FUNCTION_BLOCK FUNCTIONALITY_CONTROLLER (* Composite Function Block Type *)
  (* Standard: 61499-2 *)
  (* Version 1.0, 2019-04-04, adeel *)
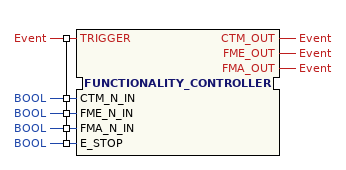
  EVENT_INPUT
    TRIGGER WITH CTM_N_IN, FME_N_IN, FMA_N_IN, E_STOP; (* Normal Execution Request *)
  END_EVENT
  EVENT_OUTPUT
    CTM_OUT; (* Execution Confirmation *)
    FME_OUT;
    FMA_OUT;
  END_EVENT
  VAR_INPUT
    CTM_N_IN : BOOL; (* Input event qualifier *)
    FME_N_IN : BOOL;
    FMA_N_IN : BOOL;
    E_STOP : BOOL;
  END_VAR
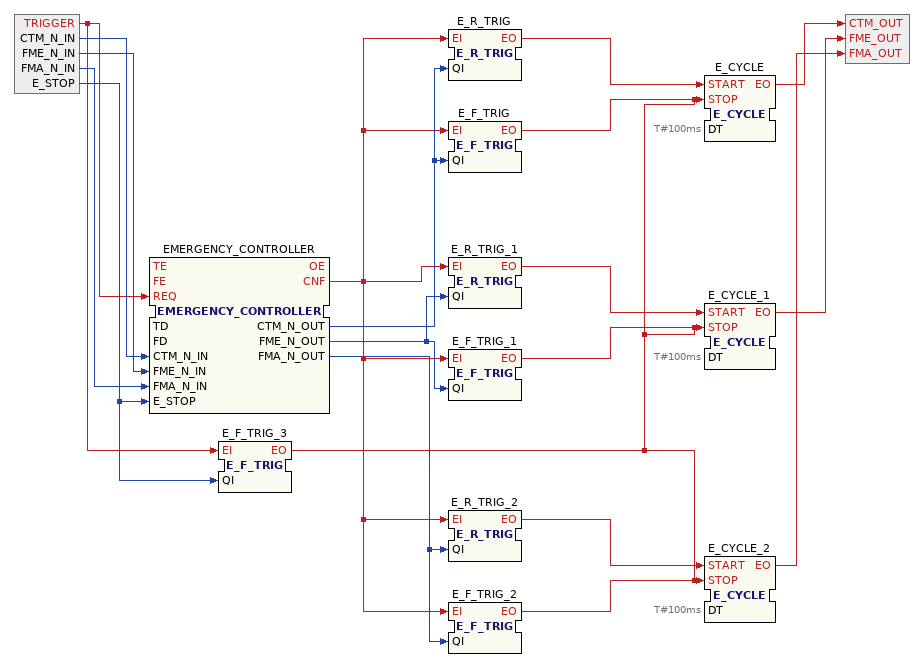
  FBS
    E_R_TRIG : E_R_TRIG;
    E_R_TRIG_1 : E_R_TRIG;
    E_R_TRIG_2 : E_R_TRIG;
    E_CYCLE : E_CYCLE(DT := T#100ms);
    E_CYCLE_1 : E_CYCLE(DT := T#100ms);
    E_CYCLE_2 : E_CYCLE(DT := T#100ms);
    E_F_TRIG : E_F_TRIG;
    E_F_TRIG_1 : E_F_TRIG;
    E_F_TRIG_2 : E_F_TRIG;
    EMERGENCY_CONTROLLER : EMERGENCY_CONTROLLER;
    E_F_TRIG_3 : E_F_TRIG;
  END_FBS
  EVENT_CONNECTIONS
    E_R_TRIG.EO TO E_CYCLE.START;
    E_F_TRIG.EO TO E_CYCLE.STOP;
    E_CYCLE.EO TO CTM_OUT;
    E_R_TRIG_1.EO TO E_CYCLE_1.START;
    E_F_TRIG_1.EO TO E_CYCLE_1.STOP;
    E_CYCLE_1.EO TO FME_OUT;
    E_R_TRIG_2.EO TO E_CYCLE_2.START;
    E_F_TRIG_2.EO TO E_CYCLE_2.STOP;
    E_CYCLE_2.EO TO FMA_OUT;
    EMERGENCY_CONTROLLER.CNF TO E_R_TRIG.EI;
    EMERGENCY_CONTROLLER.CNF TO E_F_TRIG.EI;
    EMERGENCY_CONTROLLER.CNF TO E_R_TRIG_1.EI;
    EMERGENCY_CONTROLLER.CNF TO E_F_TRIG_1.EI;
    EMERGENCY_CONTROLLER.CNF TO E_R_TRIG_2.EI;
    EMERGENCY_CONTROLLER.CNF TO E_F_TRIG_2.EI;
    TRIGGER TO EMERGENCY_CONTROLLER.REQ;
    TRIGGER TO E_F_TRIG_3.EI;
    E_F_TRIG_3.EO TO E_CYCLE.STOP;
    E_F_TRIG_3.EO TO E_CYCLE_1.STOP;
    E_F_TRIG_3.EO TO E_CYCLE_2.STOP;
  END_CONNECTIONS
  DATA_CONNECTIONS
    EMERGENCY_CONTROLLER.CTM_N_OUT TO E_R_TRIG.QI;
    EMERGENCY_CONTROLLER.CTM_N_OUT TO E_F_TRIG.QI;
    EMERGENCY_CONTROLLER.FME_N_OUT TO E_R_TRIG_1.QI;
    EMERGENCY_CONTROLLER.FME_N_OUT TO E_F_TRIG_1.QI;
    EMERGENCY_CONTROLLER.FMA_N_OUT TO E_R_TRIG_2.QI;
    EMERGENCY_CONTROLLER.FMA_N_OUT TO E_F_TRIG_2.QI;
    CTM_N_IN TO EMERGENCY_CONTROLLER.CTM_N_IN;
    FME_N_IN TO EMERGENCY_CONTROLLER.FME_N_IN;
    FMA_N_IN TO EMERGENCY_CONTROLLER.FMA_N_IN;
    E_STOP TO EMERGENCY_CONTROLLER.E_STOP;
    E_STOP TO E_F_TRIG_3.QI;
  END_CONNECTIONS
END_FUNCTION_BLOCK
